// TIA Portal V19 export
DATA_BLOCK "instWriteCanProcessImage"   // DB16
// stored: AutoNumber false, InstanceOfName WriteCanProcessImage, InstanceOfType FB
"WriteCanProcessImage"
   // VAR_OUTPUT
   //    Busy : Bool;
   //    Error : Bool;
   //    Status : DWord;
   //    Done : Bool;
   // END_VAR
   // VAR_IN_OUT
   //    CanProcessImageOutArray : Array[0..9] of Byte;
   // END_VAR
BEGIN
END_DATA_BLOCK
